FUNCTION F_IsDone : BOOL;
VAR_INPUT
	Feedback : I_CommandFeedback;
END_VAR

IF Feedback <> 0 AND_THEN Feedback.Done THEN
	F_IsDone := TRUE;
END_IF

END_FUNCTION

(* stored: Version 1.1.0.1, ProductVersion 3.1.4024.12
   POU F_IsDone: Id {620b8e3f-8997-0738-3bea-a3e66984f371}, SpecialFunc None *)
